{attribute 'qualified_only'}
VAR_GLOBAL
	//global_counter : INT := 0;
END_VAR

(* stored: Version 1.1.0.1, ProductVersion 3.1.4024.15
   GVL GVL: Id {ed47b473-7368-40f8-b818-ce840659a8dc} *)
